// TIA Portal project "Simple Ladder Logic Monitoring" (V20)

(* hardware
DEVICE "S7-1200 station_1"  S7-1200 Station
   slot 0: "Rack_0"  S7-1200 Rack  Rack  V1.0
   slot 1: "PLC_1"  CPU 1215C AC/DC/Rly  6ES7 215-1BG40-0XB0  V4.7
*)

// ===== PLC "PLC_1"  CPU 1215C AC/DC/Rly =====

VAR_GLOBAL   // PLC tag table "Default tag table"
   "Tag_1" AT %Q0.0 : Bool;
   "Light 4" AT %Q0.4 : Bool;
   "Switch 4" AT %I0.3 : Bool;
END_VAR

VAR_GLOBAL   // PLC tag table "Tag table_1"
   "Switch 1" AT %I0.0 : Bool;
   "Switch 2" AT %I0.1 : Bool;
   "Switch 3" AT %I0.2 : Bool;
   "Pot 1" AT %QW1 : Int;
   "Pot 2" AT %QW2 : Int;
   "Light 1" AT %M0.0 : Bool;
   "Light 2" AT %M0.1 : Bool;
   "Light 3" AT %M0.2 : Bool;
   "Button HMI" AT %M0.4 : Bool;   // for hmi
END_VAR

ORGANIZATION_BLOCK "Main"   // OB1, LAD, ProgramCycle
TITLE = "Main Program Sweep (Cycle)"
{ S7_Optimized_Access := 'TRUE' }
VERSION : 0.1
   VAR_INPUT
      Initial_Call : Bool;   // Initial call of this OB
      Remanence : Bool;   // =True, if remanent data are available
   END_VAR
BEGIN

REGION Network 1
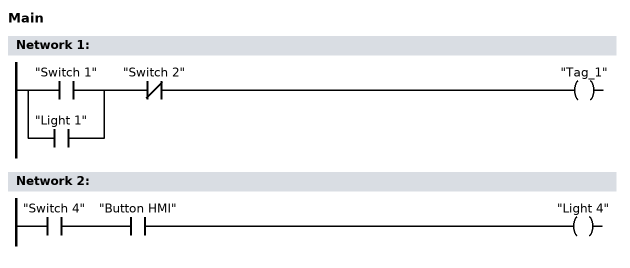
   RUNG wire#powerrail
      Contact( "Switch 1" )
      wire#w1
      I_Contact( "Switch 2" )
      Coil( "Tag_1" )
   END_RUNG
   RUNG wire#powerrail
      Contact( "Light 1" )
   END_RUNG wire#w1
   // the same network as SCL:
   "Tag_1" := ("Switch 1" OR "Light 1") AND NOT "Switch 2";
END_REGION

REGION Network 2
   RUNG wire#powerrail
      Contact( "Switch 4" )
      Contact( "Button HMI" )
      Coil( "Light 4" )
   END_RUNG
   // the same network as SCL:
   "Light 4" := "Switch 4" AND "Button HMI";
END_REGION
END_ORGANIZATION_BLOCK